RoboDK station: solar_tracker.rdk

Station solar_tracker (saved by RoboDK 5.9.6). Poses are relative to the parent item; angles as X-Y-Z fixed-axis rotations.
  - frame Azimuth at (0, 0, 0) mm
    - frame Elevation at (0, 0, 1000) mm, rotated rx 90 ry 0 rz 90 deg
